FUNCTION_BLOCK Test_TExecutionWhenBusy_Start_RaisesEvent EXTENDS TUnitTestbase
VAR
    Execution : TExecution;
    Execution_EventHandler : TExecution_EventHandler;
END_VAR

// Setup...
Execution.FB_init(
    bInitRetains := FALSE,
    bInCopyCode  := FALSE);
Execution_EventHandler.FB_init(
    bInitRetains := FALSE,
    bInCopyCode  := FALSE);

// link handler to common execution events...
GlobalEvents.Event_OnAbort.ClearEventHandlers().AddEventHandler(Execution_EventHandler);
GlobalEvents.Event_OnError.ClearEventHandlers().AddEventHandler(Execution_EventHandler);

// Test...
Execution.Start(); // sets Starting

Execution.Start(); // raises error event

Assertion.AssertEquals_BOOL(
    Expected := TRUE,
    Actual   := Execution_EventHandler.FailedEventRaised,
    VariableName  := 'EventHandler.FailedEventRaised');
    
    
TestFinished();

END_FUNCTION_BLOCK

(* stored: Version 1.1.0.1, ProductVersion 3.1.4024.4
   POU Test_TExecutionWhenBusy_Start_RaisesEvent: Id {cc576e06-690c-4823-83da-e4831a38e124}, SpecialFunc None *)
